  def norm_to_gripper(value_norm):
      value_gripper = (value_norm / 100) * 255
      return ceil(value_gripper)
  end

  def rq_get_position():
      return rq_current_pos_norm()
  end

  def rq_gripper_led_on(gripper_socket="1"):
      rq_set_var("LBP",0, gripper_socket)
  end

  def rq_gripper_led_off(gripper_socket="1"):
      rq_set_var("LBP",1, gripper_socket)
      rq_set_var("LRD",0, gripper_socket)
      rq_set_var("LBL",0, gripper_socket)
      rq_set_var("LGN",0, gripper_socket)
  end

  def rq_gripper_led_force_red(gripper_socket="1"):
      rq_set_var("LBP",1, gripper_socket)
      rq_set_var("LRD",1, gripper_socket)
      rq_set_var("LBL",0, gripper_socket)
      rq_set_var("LGN",0, gripper_socket)
  end

  def rq_gripper_led_force_blue(gripper_socket="1"):
      rq_set_var("LBP",1, gripper_socket)
      rq_set_var("LRD",0, gripper_socket)
      rq_set_var("LBL",1, gripper_socket)
      rq_set_var("LGN",0, gripper_socket)
  end

  def rq_gripper_led_force_green(gripper_socket="1"):
      rq_set_var("LBP",1, gripper_socket)
      rq_set_var("LRD",0, gripper_socket)
      rq_set_var("LBL",0, gripper_socket)
      rq_set_var("LGN",1, gripper_socket)
  end

  def rq_gripper_led_force_purple(gripper_socket="1"):
      rq_set_var("LBP",1, gripper_socket)
      rq_set_var("LRD",1, gripper_socket)
      rq_set_var("LBL",1, gripper_socket)
      rq_set_var("LGN",0, gripper_socket)
  end

  ############################################
  # mm/inches functions
  ############################################
  gripper_closed_norm = [100, 100, 100, 100]
  gripper_open_norm = [0, 0, 0, 0]
  gripper_closed_mm = [0, 0, 0, 0]
  gripper_open_mm = [50, 50, 50, 50]

  def rq_current_pos_mm(gripper_socket=1):
      pos_gripper = rq_current_pos(gripper_socket)
      pos_mm = gripper_to_mm(pos_gripper, gripper_socket)
      return round_value_2_dec(pos_mm)
  end

  def rq_current_pos_inches(gripper_socket=1):
      pos_gripper = rq_current_pos(gripper_socket)
      pos_mm = gripper_to_mm(pos_gripper, gripper_socket)
      pos_in = pos_mm / 25.4
      return round_value_2_dec(pos_in)
  end

  def rq_move_mm(pos_mm, gripper_socket=1):
      pos_gripper = mm_to_gripper(pos_mm, gripper_socket)
      rq_move(pos_gripper, gripper_socket)
  end

  def rq_move_and_wait_mm(pos_mm, gripper_socket=1):
      pos_gripper = mm_to_gripper(pos_mm, gripper_socket)
      rq_move_and_wait(pos_gripper, gripper_socket)
  end

  def rq_move_inches(pos_in, gripper_socket=1):
      pos_mm = pos_in * 25.4
      rq_move_mm(pos_mm, gripper_socket)
  end

  def rq_move_and_wait_inches(pos_in, gripper_socket=1):
      pos_mm = pos_in * 25.4
      rq_move_and_wait_mm(pos_mm, gripper_socket)
  end

  def get_closed_norm(gripper_socket):
      return gripper_closed_norm[gripper_socket - 1]
  end

  def get_open_norm(gripper_socket):
      return gripper_open_norm[gripper_socket - 1]
  end

  def get_closed_mm(gripper_socket):
      return gripper_closed_mm[gripper_socket - 1]
  end

  def get_open_mm(gripper_socket):
      return gripper_open_mm[gripper_socket - 1]
  end

  def set_closed_norm(closed_norm, gripper_socket):
      gripper_closed_norm[gripper_socket - 1] = closed_norm
  end

  def set_open_norm(open_norm, gripper_socket):
      gripper_open_norm[gripper_socket - 1] = open_norm
  end

  def set_closed_mm(closed_mm, gripper_socket):
      gripper_closed_mm[gripper_socket - 1] = closed_mm
  end

  def set_open_mm(open_mm, gripper_socket):
      gripper_open_mm[gripper_socket - 1] = open_mm
  end

  def gripper_to_mm(value_gripper, gripper_socket):
      closed_norm = get_closed_norm(gripper_socket)
      open_norm = get_open_norm(gripper_socket)
      closed_mm = get_closed_mm(gripper_socket)
      open_mm = get_open_mm(gripper_socket)

      value_norm = (value_gripper / 255) * 100

      slope = (closed_mm - open_mm) / (closed_norm - open_norm)
      value_mm = slope * (value_norm - closed_norm) + closed_mm

      if (value_mm > open_mm):
          value_mm_limited = open_mm
      elif (value_mm < closed_mm):
          value_mm_limited = closed_mm
      else:
          value_mm_limited = value_mm
      end

      return value_mm_limited
  end

  def mm_to_gripper(value_mm, gripper_socket):
      closed_norm = get_closed_norm(gripper_socket)
      open_norm = get_open_norm(gripper_socket)
      closed_mm = get_closed_mm(gripper_socket)
      open_mm = get_open_mm(gripper_socket)

      slope = (closed_norm - open_norm) / (closed_mm - open_mm)
      value_norm = (value_mm - closed_mm) * slope + closed_norm

      value_gripper = value_norm * 255 / 100

      if (value_gripper > 255):
          value_gripper_limited = 255
      elif (value_gripper < 0):
          value_gripper_limited = 0
      else:
          value_gripper_limited = round_value(value_gripper)
      end

      return value_gripper_limited
  end

  def round_value(value):
      value_mod = value % 1

      if(value_mod < 0.5):
          return floor(value)
      else:
          return ceil(value)
      end
  end

  def round_value_2_dec(value):
      value_x_100 = value * 100
      value_x_100_rounded = round_value(value_x_100)
      return value_x_100_rounded / 100
  end

  def clear_socket_buffer(gripper_socket="1", read_timeout = 0.1):
      rq_comm_clear_socket_buffer_enabled[rq_socket_to_index(gripper_socket)] = True
  end

  def rq_gripper_id_to_ascii(gripper_id):
      if(gripper_id == "1"):
          return 57
      elif(gripper_id == "2"):
          return 50
      elif(gripper_id == "3"):
          return 51
      elif(gripper_id == "4"):
          return 52
      end
  end

  def scale(value, rawRange, scaledRange):
      def computeSlope(inputRange, outputRange):
          outputRangeDelta = outputRange[1] - outputRange[0]
          inputRangeDelta = inputRange[1] - inputRange[0]

          if (inputRangeDelta == 0):
              return 0
          else:
              return outputRangeDelta / inputRangeDelta
          end
      end

      def computeIntercept(slope, inputRange, outputRange):
          return outputRange[0] - (slope * inputRange[0])
      end

      def clipScaledValue(outputScaledValue, outputRange):
          if (outputRange[0] < outputRange[1]):
              return clipWhenLowerLimitIsLessThanHigher(outputScaledValue, outputRange)
          else:
              return clipWhenLowerLimitIsGreaterThanHigherLimit(outputScaledValue, outputRange)
          end
      end

      def clipWhenLowerLimitIsGreaterThanHigherLimit(outputScaledValue, outputRange):
          if (outputScaledValue < outputRange[1]):
              return outputRange[1]
          elif (outputScaledValue > outputRange[0]):
              return outputRange[0]
          else:
              return outputScaledValue
          end
      end

      def clipWhenLowerLimitIsLessThanHigher(outputScaledValue, outputRange):
          if (outputScaledValue < outputRange[0]):
              return outputRange[0]
          elif (outputScaledValue > outputRange[1]):
              return outputRange[1]
          else:
              return outputScaledValue
          end
      end

      slope = computeSlope(rawRange, scaledRange)
      intercept = computeIntercept(slope, rawRange, scaledRange)
      scaledValue = slope * value + intercept
      return clipScaledValue(scaledValue, scaledRange)
  end

  def limit(value, range):
      return scale(value, range, range)
  end


  rq_init_comm_if_connected(9, "1")
  rq_init_comm_if_connected(2, "2")
  rq_init_comm_if_connected(3, "3")
  rq_init_comm_if_connected(4, "4")
  rq_print_connected_grippers()
  rq_gripper_communication_thread = run rq_gripper_communication()
  set_closed_norm(100.0, 1)
  set_open_norm(0.0, 1)
  set_closed_mm(0.0, 1)
  set_open_mm(50.0, 1)
  set_closed_norm(100.0, 2)
  set_open_norm(0.0, 2)
  set_closed_mm(0.0, 2)
  set_open_mm(50.0, 2)
  set_closed_norm(100.0, 3)
  set_open_norm(0.0, 3)
  set_closed_mm(0.0, 3)
  set_open_mm(50.0, 3)
  set_closed_norm(100.0, 4)
  set_open_norm(0.0, 4)
  set_closed_mm(0.0, 4)
  set_open_mm(50.0, 4)
  rq_current_limit_enabled = False
  while(not rq_gripper_communication_thread_started):
      sleep(0.008)
  end
  # end: URCap Installation Node
  $ 1 "BeforeStart"
  # begin: URCap Program Node
  #   Source: Robotiq_Grippers, 1.8.9.14887, Robotiq Inc.
  #   Type: Gripper Activate
  $ 2 "Gripper Activate"

  kill rq_gripper_communication_thread
  rq_gripper_communication_thread_started = False
  rq_close_gripper_socket("1")
  rq_close_gripper_socket("2")
  rq_close_gripper_socket("3")
  rq_close_gripper_socket("4")

  rq_init_comm_if_connected(9, "1")
  rq_init_comm_if_connected(2, "2")
  rq_init_comm_if_connected(3, "3")
  rq_init_comm_if_connected(4, "4")
  rq_print_connected_grippers()
  rq_gripper_communication_thread = run rq_gripper_communication()

  while(not rq_gripper_communication_thread_started):
      sleep(0.008)
  end

  rq_set_max_current_for_all_grippers()

  reset_and_activate = False

  rq_activate_all_grippers(False)
  # end: URCap Program Node
  # begin: URCap Program Node
  #   Source: Robotiq_Grippers, 1.8.9.14887, Robotiq Inc.
  #   Type: Gripper
  $ 3 "Gripper Open (1)"
  if not(gripper_connected[0]):
    popup("Gripper 1 must be connected to run this program.", "No connection", False, True, True)
  end
  if not(rq_is_gripper_activated("1")):
    popup("Gripper 1 is not activated. Go to Installation tab > Gripper to activate it and run the program again.", "Not activated", False, True, True)
  end
  rq_set_pos_spd_for(0, 255, 0, "1")
  rq_wait_pos_spe_for_request(0, 255, 0, "1")
  rq_go_to("1")
  rq_wait("1")
  # end: URCap Program Node
  $ 4 "MoveJ"
  $ 5 "Rest" "breakAfter"
  movej(get_inverse_kin(p[-.112987348259, -.297700236568, .156260077323, -2.222194308145, -2.218522570111, -.000095127165], qnear=[-1.5707963267948966, -1.5707724730123083, -1.570783917103662, -1.570760075246131, 1.5707907676699604, 1.570730805396848]), a=1.3962634015954636, v=1.0471975511965976)
  $ 6 "MoveJ"
  $ 7 "exit_picking" "breakAfter"
  movej(get_inverse_kin(p[.158290115728, -.354639829756, .152934438952, -.013774424009, 3.096323764078, -.057423310476], qnear=[-0.8629029432879847, -1.823266331349508, -1.3230798880206507, -1.5076640287982386, 1.5825906991958618, 0.6976197361946106]), a=1.3962634015954636, v=1.0471975511965976)
  $ 8 "MoveJ"
  $ 9 "Pick_Up" "breakAfter"
  movej(get_inverse_kin(p[.158292635212, -.354628935188, .081389339757, -.013605428178, 3.096205221041, -.057452890653], qnear=[-0.8629267851458948, -1.8724725882159632, -1.6003153959857386, -1.1811254660235804, 1.5829143524169922, 0.6980634927749634]), a=1.3962634015954636, v=1.0471975511965976)
  $ 10 "MoveJ"
  $ 11 "exit_picking" "breakAfter"
  movej(get_inverse_kin(p[.158290115728, -.354639829756, .152934438952, -.013774424009, 3.096323764078, -.057423310476], qnear=[-0.8629029432879847, -1.823266331349508, -1.3230798880206507, -1.5076640287982386, 1.5825906991958618, 0.6976197361946106]), a=1.3962634015954636, v=1.0471975511965976)
  $ 12 "MoveJ"
  $ 13 "drop_entry" "breakAfter"
  movej(get_inverse_kin(p[-.112857914387, -.292299128717, .116006763882, 2.220836260040, 2.218808085372, -.006301776434], qnear=[-1.5702689329730433, -1.5589354673968714, -1.7748406569110315, -1.3729618231402796, 1.5707064867019653, 1.5707188844680786]), a=1.3962634015954636, v=1.0471975511965976)
  $ 14 "MoveJ"
  $ 15 "drop" "breakAfter"
  movej(get_inverse_kin(p[-.112615056925, -.302416342261, .012836420119, 2.219842457995, 2.220208331981, -.006547852640], qnear=[-1.5693705717669886, -1.7935569922076624, -2.0517805258380335, -0.8614938894854944, 1.5709584951400757, 1.5710548162460327]), a=1.3962634015954636, v=1.0471975511965976)
  # begin: URCap Program Node
  #   Source: Robotiq_Grippers, 1.8.9.14887, Robotiq Inc.
  #   Type: Gripper Activate
  $ 16 "Gripper Activate"

  kill rq_gripper_communication_thread
  rq_gripper_communication_thread_started = False
  rq_close_gripper_socket("1")
  rq_close_gripper_socket("2")
  rq_close_gripper_socket("3")
  rq_close_gripper_socket("4")

  rq_init_comm_if_connected(9, "1")
  rq_init_comm_if_connected(2, "2")
  rq_init_comm_if_connected(3, "3")
  rq_init_comm_if_connected(4, "4")
  rq_print_connected_grippers()
  rq_gripper_communication_thread = run rq_gripper_communication()

  while(not rq_gripper_communication_thread_started):
      sleep(0.008)
  end

  rq_set_max_current_for_all_grippers()

  reset_and_activate = False

  rq_activate_all_grippers(False)
  # end: URCap Program Node
  $ 17 "P≔Pick_Up"
  global P=p[.158292635212, -.354628935188, .081389339757, -.013605428178, 3.096205221041, -.057452890653]
  $ 18 "D≔drop"
  global D=p[-.112615056925, -.302416342261, .012836420119, 2.219842457995, 2.220208331981, -.006547852640]
  $ 19 "distance≔0.024"
  global distance=0.024
  $ 20 "Popup: fine prestart"
  popup("fine prestart", "Message", False, False, blocking=True)
  while (True):
    $ 21 "Robot Program"
    $ 22 "Loop 4 times"
    Loop_2 = 0
    while (Loop_2 < 4):
      $ 23 "MoveJ"
      $ 24 "drop_entry" "breakAfter"
      movej(get_inverse_kin(p[-.112857914387, -.292299128717, .116006763882, 2.220836260040, 2.218808085372, -.006301776434], qnear=[-1.5702689329730433, -1.5589354673968714, -1.7748406569110315, -1.3729618231402796, 1.5707064867019653, 1.5707188844680786]), a=1.3962634015954636, v=1.0471975511965976)
      $ 25 "MoveJ"
      $ 26 "exit_picking" "breakAfter"
      movej(get_inverse_kin(p[.158290115728, -.354639829756, .152934438952, -.013774424009, 3.096323764078, -.057423310476], qnear=[-0.8629029432879847, -1.823266331349508, -1.3230798880206507, -1.5076640287982386, 1.5825906991958618, 0.6976197361946106]), a=1.3962634015954636, v=1.0471975511965976)
      $ 27 "MoveL"
      $ 28 "P" "breakAfter"
      movel(pose_trans(p[0.0,0.0,0.0,0.0,0.0,0.0], P), a=1.2, v=0.25)
      # begin: URCap Program Node
      #   Source: Robotiq_Grippers, 1.8.9.14887, Robotiq Inc.
      #   Type: Gripper
      $ 29 "Gripper Close (1)"
      if not(gripper_connected[0]):
        popup("Gripper 1 must be connected to run this program.", "No connection", False, True, True)
      end
      if not(rq_is_gripper_activated("1")):
        popup("Gripper 1 is not activated. Go to Installation tab > Gripper to activate it and run the program again.", "Not activated", False, True, True)
      end
      rq_set_pos_spd_for(255, 0, 0, "1")
      rq_wait_pos_spe_for_request(255, 0, 0, "1")
      rq_go_to("1")
      rq_wait("1")
      # end: URCap Program Node
      $ 30 "MoveL"
      $ 31 "exit_picking" "breakAfter"
      movel(p[.158290115728, -.354639829756, .152934438952, -.013774424009, 3.096323764078, -.057423310476], a=1.2, v=0.25)
      $ 32 "MoveL"
      $ 33 "drop_entry" "breakAfter"
      movel(p[-.112857914387, -.292299128717, .116006763882, 2.220836260040, 2.218808085372, -.006301776434], a=1.2, v=0.25)
      $ 34 "MoveL"
      $ 35 "D" "breakAfter"
      movel(pose_trans(p[0.0,0.0,0.0,0.0,0.0,0.0], D), a=1.2, v=0.25)
      # begin: URCap Program Node
      #   Source: Robotiq_Grippers, 1.8.9.14887, Robotiq Inc.
      #   Type: Gripper
      $ 36 "Gripper Open (1)"
      if not(gripper_connected[0]):
        popup("Gripper 1 must be connected to run this program.", "No connection", False, True, True)
      end
      if not(rq_is_gripper_activated("1")):
        popup("Gripper 1 is not activated. Go to Installation tab > Gripper to activate it and run the program again.", "Not activated", False, True, True)
      end
      rq_set_pos_spd_for(0, 0, 0, "1")
      rq_wait_pos_spe_for_request(0, 0, 0, "1")
      rq_go_to("1")
      rq_wait("1")
      # end: URCap Program Node
      $ 37 "P[2]=P[2]-distance"
      P[2]=P[2]-distance
      $ 38 "D[2]=D[2]+(distance+0.005)"
      D[2]=D[2]+(distance+0.005)
      Loop_2 = Loop_2 + 1
    end
    $ 39 "If Loop_2≟4"
    global thread_flag_39=0
    thread Thread_if_39():
      $ 40 "D≔drop"
      global D=p[-.112615056925, -.302416342261, .012836420119, 2.219842457995, 2.220208331981, -.006547852640]
      $ 41 "P≔Pick_Up"
      global P=p[.158292635212, -.354628935188, .081389339757, -.013605428178, 3.096205221041, -.057452890653]
      $ 42 "Popup: Fine impilamento"
      popup("Fine impilamento", "Message", False, False, blocking=True)
      thread_flag_39 = 1
    end
    if (Loop_2 == 4):
      global thread_handler_39=run Thread_if_39()
      while (thread_flag_39 == 0):
        if not(Loop_2 == 4):
          kill thread_handler_39
          thread_flag_39 = 2
        else:
          sync()
        end
      end
    else:
      thread_flag_39 = 2
    end
  end
end
